// TIA Portal V17 export
// export: Created 2023-12-05T13:40:23.2775164Z, ExportSetting WithDefaults, DisplayName Totally Integrated Automation Portal, DisplayVersion V17, DisplayName TIA Portal Openness, DisplayVersion V17, DisplayName TIA Portal Version Control Interface, DisplayVersion V17, DisplayName SINAMICS Startdrive Advanced, DisplayVersion V17, DisplayName SINAMICS Startdrive G130, G150, S120, S150, SINAMICS MV, S210, DisplayVersion V17, DisplayName SINAMICS Startdrive G110M, G120, G120C, G120D, G120P, G115D, DisplayVersion V17, DisplayName STEP 7 Professional, DisplayVersion V17, DisplayName STEP 7 Safety, DisplayVersion V17, DisplayName WinCC Professional, DisplayVersion V17
FUNCTION "FC535 ACSD_V5_1_7 Alarms" : Void   // FC535, LAD
{ S7_Optimized_Access := 'TRUE' }
VERSION : 0.1
// LG 23.03.2023 => Created block
// stored: AutoNumber false, IsIECCheckEnabled false, SetENOAutomatically false, UDAEnableTagReadback false
   VAR_INPUT
      AckStep : Bool;
      "SB DB" : Int;
      "Alarm DB" : Int;
      "Alarm Offset" : Int;
   END_VAR
   VAR_TEMP
      "SB DBW" : Word;
      "AL DBW" : Word;
      "TR DBW" : Word;
   END_VAR
BEGIN

NETWORK
TITLE = Initialization
      L     #"SB DB";
      T     #"SB DBW";
      L     #"Alarm DB";
      T     #"AL DBW";
      L     #"Alarm Offset";
      SLD   3;
      LAR1;

NETWORK
TITLE = Cylinder faults
      CLR;
      OPN   DB [#"SB DBW"];
      L     %DBB70;
      OPN   DB [#"AL DBW"];
      T     DBB [AR1, P#0.0];

NETWORK
TITLE = Cylinder faults
// DBX169.0 - Clean Hotplates
      CLR;
      OPN   DB [#"SB DBW"];
      A     %DBX71.0;
      OPN   DB [#"AL DBW"];
      =     DBX [AR1, P#1.0];

NETWORK
TITLE = RCFaults
      A     #AckStep;
      JCN   eno;
      CLR;
      OPN   DB [#"SB DBW"];
      L     %DBB74;
      OPN   DB [#"AL DBW"];
      T     DBB [AR1, P#2.0];
eno:  NOP   0;

NETWORK
TITLE = Faults .0
      CLR;
      OPN   DB [#"SB DBW"];
      A     %DBX76.0;
      OPN   DB [#"AL DBW"];
      =     DBX [AR1, P#4.0];

NETWORK
TITLE = Faults .1
      CLR;
      OPN   DB [#"SB DBW"];
      A     %DBX76.1;
      OPN   DB [#"AL DBW"];
      =     DBX [AR1, P#4.1];

NETWORK
TITLE = Faults .2
      CLR;
      OPN   DB [#"SB DBW"];
      A     %DBX76.2;
      OPN   DB [#"AL DBW"];
      =     DBX [AR1, P#4.2];

NETWORK
TITLE = Faults .3
      CLR;
      OPN   DB [#"SB DBW"];
      A     %DBX76.3;
      OPN   DB [#"AL DBW"];
      =     DBX [AR1, P#4.3];

NETWORK
TITLE = Faults .4
      CLR;
      OPN   DB [#"SB DBW"];
      A     %DBX76.4;
      OPN   DB [#"AL DBW"];
      =     DBX [AR1, P#4.4];
END_FUNCTION
